FUNCTION_BLOCK InfoDataAdsAoEDC EXTENDS InfoDataAdsAoE
VAR
	_dcOutputShift AT %I* :   DINT;
	_dcInputShift AT %I* :   DINT;
END_VAR

PROPERTY AdsAddr : AMSADDR
GET
AdsAddr := _AdsAddr;
END_GET
END_PROPERTY

END_FUNCTION_BLOCK

(* stored: Version 1.1.0.1, ProductVersion 3.1.4024.9
   POU InfoDataAdsAoEDC: Id {b6f940a7-08c7-061c-3fc6-7a045f0f3fb7}, SpecialFunc None
   Property AdsAddr: Id {0de6a5f3-7e77-0386-28ed-d973d673b22c}
   Get Get: Id {010290d8-365a-0469-2f54-20666985ad18} *)
